// TIA Portal V16 export
// export: Created 2023-01-04T15:44:09.1719163Z, ExportSetting WithDefaults, DisplayName Totally Integrated Automation Portal, DisplayVersion V16, DisplayName TIA Portal Version Control Interface, DisplayVersion V16, DisplayName TIA Portal Openness, DisplayVersion V16, DisplayName STEP 7 Professional, DisplayVersion V16, DisplayName STEP 7 Safety, DisplayVersion V16, DisplayName WinCC Advanced, DisplayVersion V16
DATA_BLOCK "Filling_Logic_DB"   // DB4
VERSION : 0.1
// stored: AutoNumber true, DBAccessibleFromOPCUA true, InstanceOfName Filling_Logic, InstanceOfType FB
"Filling_Logic"
   // VAR_INPUT
   //    PS2_Filling_Station : Bool;
   //    FIC_B102 : Int;
   //    Liquid_AorB_in_Bottle_ml : Real;
   //    Liquid_AorB_pct : Int;
   //    PTRIG3 : Bool;
   //    PTRIG2 : Bool;
   //    Wait_to_fill : Time;
   // END_VAR
   // VAR_OUTPUT
   //    Outlet_of_tanks : Bool;
   //    Flow_ml_per_sec : Real;
   //    PTRIG1 : Bool;
   //    FillingData_LiqAorB_ml : Real;
   // END_VAR
BEGIN
END_DATA_BLOCK
